(* PLC project Tc2_MC2.MC_MoveContinuousAbsolute Demo, tc3-libraries-kb TwinCAT 3.1 *)
(* stored: creationDateTime 2026-05-21T00:00:00, modificationDateTime 2026-05-21T00:00:00 *)

PROGRAM P_Demo_MC_MoveContinuousAbsolute
  VAR
    fbStraightCut : MC_MoveContinuousAbsolute;
    fbHaltSafety : MC_Halt;
    axisLaserHead : AXIS_REF;
    rtCutTrig : R_TRIG;
    rtSafetyHalt : R_TRIG;
    bStartStraight : BOOL := FALSE;
    bEmergencyStop : BOOL := FALSE;
    bInArc : BOOL;
    bSafetyHaltDone : BOOL;
    nErrorID : UDINT;
  END_VAR

// =============================================================================
// 场景：激光切割机 — 直线段切到 100 mm 时不要停（停了会出过烧痕），保持
//       200 mm/s 进入下一段圆弧。EndVelocity = 200 是关键。
// 价值：业务给绝对终点 + 终末速度两个量，FB 自动算减速曲线让到位时速度恰好。
// 验证：bStartStraight := TRUE → 看 ActPos 加速到 1000 mm/s 走到 100 mm，
//       到位时 ActVelo ≈ 200，bInArc 置 TRUE。bEmergencyStop := TRUE → 兜底停车。
// =============================================================================

rtCutTrig(CLK := bStartStraight);
rtSafetyHalt(CLK := bEmergencyStop);

fbStraightCut(
    Execute       := rtCutTrig.Q,
    Position      := 100.0,
    Velocity      := 1000.0,
    EndVelocity   := 200.0,
    Acceleration  := 5000.0,
    Deceleration  := 5000.0,
    Jerk          := 50000.0,
    BufferMode    := MC_Buffered,
    Axis          := axisLaserHead,
    InEndVelocity => bInArc,
    ErrorID       => nErrorID
);

fbHaltSafety(
    Execute      := rtSafetyHalt.Q,
    Deceleration := 10000.0,
    Jerk         := 100000.0,
    Axis         := axisLaserHead,
    Done         => bSafetyHaltDone
);
END_PROGRAM
